// TIA Portal V20 export
ORGANIZATION_BLOCK "MainOB"   // OB125, LAD, ProgramCycle
TITLE = "Main Program Sweep (Cycle)"
{ S7_Optimized_Access := 'TRUE' }
// stored: SetENOAutomatically false
   VAR_INPUT
      Initial_Call : Bool;   // Initial call of this OB
      Remanence : Bool;   // =True, if remanent data are available
   END_VAR
BEGIN

REGION Network 1
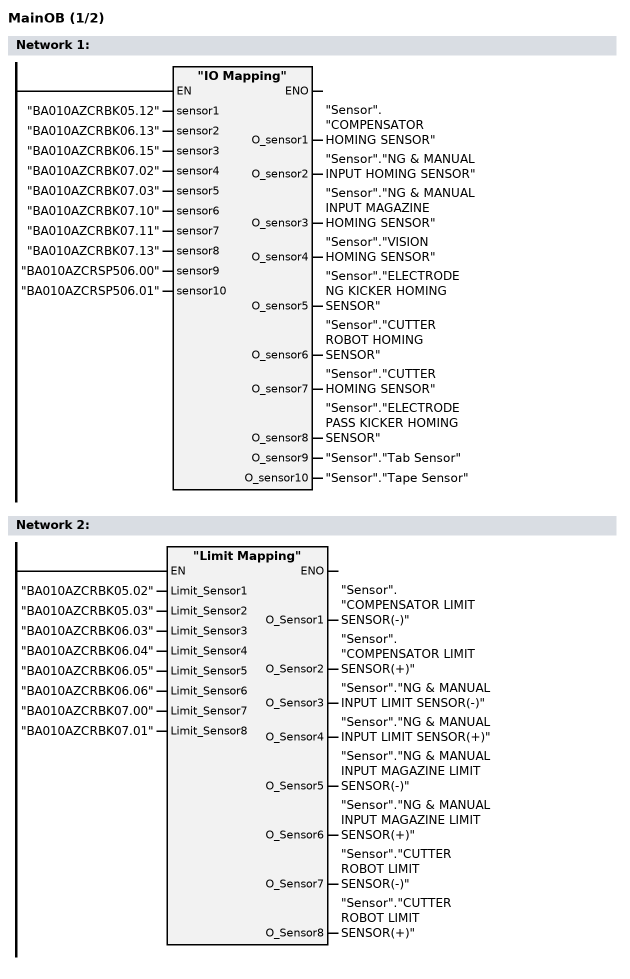
   "IO Mapping"(sensor1 := "BA010AZCRBK05.12",
                sensor2 := "BA010AZCRBK06.13",
                sensor3 := "BA010AZCRBK06.15",
                sensor4 := "BA010AZCRBK07.02",
                sensor5 := "BA010AZCRBK07.03",
                sensor6 := "BA010AZCRBK07.10",
                sensor7 := "BA010AZCRBK07.11",
                sensor8 := "BA010AZCRBK07.13",
                sensor9 := "BA010AZCRSP506.00",
                sensor10 := "BA010AZCRSP506.01",
                O_sensor1 => "Sensor"."COMPENSATOR HOMING SENSOR",
                O_sensor2 => "Sensor"."NG & MANUAL INPUT HOMING SENSOR",
                O_sensor3 => "Sensor"."NG & MANUAL INPUT MAGAZINE HOMING SENSOR",
                O_sensor4 => "Sensor"."VISION HOMING SENSOR",
                O_sensor5 => "Sensor"."ELECTRODE NG KICKER HOMING SENSOR",
                O_sensor6 => "Sensor"."CUTTER ROBOT HOMING SENSOR",
                O_sensor7 => "Sensor"."CUTTER HOMING SENSOR",
                O_sensor8 => "Sensor"."ELECTRODE PASS KICKER HOMING SENSOR",
                O_sensor9 => "Sensor"."Tab Sensor",
                O_sensor10 => "Sensor"."Tape Sensor");
END_REGION

REGION Network 2
   "Limit Mapping"(Limit_Sensor1 := "BA010AZCRBK05.02",
                   Limit_Sensor2 := "BA010AZCRBK05.03",
                   Limit_Sensor3 := "BA010AZCRBK06.03",
                   Limit_Sensor4 := "BA010AZCRBK06.04",
                   Limit_Sensor5 := "BA010AZCRBK06.05",
                   Limit_Sensor6 := "BA010AZCRBK06.06",
                   Limit_Sensor7 := "BA010AZCRBK07.00",
                   Limit_Sensor8 := "BA010AZCRBK07.01",
                   O_Sensor1 => "Sensor"."COMPENSATOR LIMIT SENSOR(-)",
                   O_Sensor2 => "Sensor"."COMPENSATOR LIMIT SENSOR(+)",
                   O_Sensor3 => "Sensor"."NG & MANUAL INPUT LIMIT SENSOR(-)",
                   O_Sensor4 => "Sensor"."NG & MANUAL INPUT LIMIT SENSOR(+)",
                   O_Sensor5 => "Sensor"."NG & MANUAL INPUT MAGAZINE LIMIT SENSOR(-)",
                   O_Sensor6 => "Sensor"."NG & MANUAL INPUT MAGAZINE LIMIT SENSOR(+)",
                   O_Sensor7 => "Sensor"."CUTTER ROBOT LIMIT SENSOR(-)",
                   O_Sensor8 => "Sensor"."CUTTER ROBOT LIMIT SENSOR(+)");
END_REGION

REGION Network 3
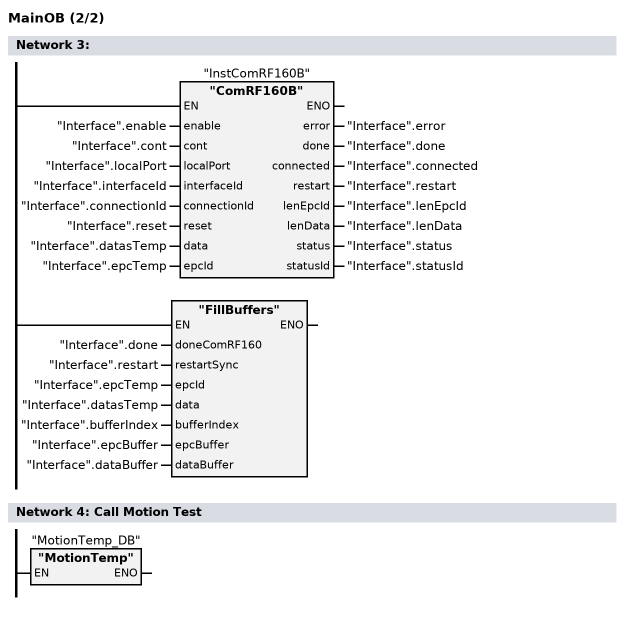
   RUNG wire#powerrail
      "InstComRF160B"(enable := "Interface".enable, cont := "Interface".cont, localPort := "Interface".localPort, interfaceId := "Interface".interfaceId, connectionId := "Interface".connectionId, reset := "Interface".reset, data := "Interface".datasTemp, epcId := "Interface".epcTemp, error => "Interface".error, done => "Interface".done, connected => "Interface".connected, restart => "Interface".restart, lenEpcId => "Interface".lenEpcId, lenData => "Interface".lenData, status => "Interface".status, statusId => "Interface".statusId)
   END_RUNG
   RUNG wire#powerrail
      "FillBuffers"(doneComRF160 := "Interface".done, restartSync := "Interface".restart, epcId := "Interface".epcTemp, data := "Interface".datasTemp, bufferIndex := "Interface".bufferIndex, epcBuffer := "Interface".epcBuffer, dataBuffer := "Interface".dataBuffer)
   END_RUNG
   // the same network as SCL:
   "InstComRF160B"(enable := "Interface".enable,   // "ComRF160B"
                   cont := "Interface".cont,
                   localPort := "Interface".localPort,
                   interfaceId := "Interface".interfaceId,
                   connectionId := "Interface".connectionId,
                   reset := "Interface".reset,
                   data := "Interface".datasTemp,
                   epcId := "Interface".epcTemp,
                   error => "Interface".error,
                   done => "Interface".done,
                   connected => "Interface".connected,
                   restart => "Interface".restart,
                   lenEpcId => "Interface".lenEpcId,
                   lenData => "Interface".lenData,
                   status => "Interface".status,
                   statusId => "Interface".statusId);
   "FillBuffers"(doneComRF160 := "Interface".done,
                 restartSync := "Interface".restart,
                 epcId := "Interface".epcTemp,
                 data := "Interface".datasTemp,
                 bufferIndex := "Interface".bufferIndex,
                 epcBuffer := "Interface".epcBuffer,
                 dataBuffer := "Interface".dataBuffer);
END_REGION

REGION Network 4: Call Motion Test
   RUNG wire#powerrail
      "MotionTemp_DB"()
   END_RUNG
   // the same network as SCL:
   "MotionTemp_DB"();   // "MotionTemp"
END_REGION
END_ORGANIZATION_BLOCK
